{attribute 'linkalways'} 
{attribute 'no_explicit_call' := 'This FB is a CLASS and must be accessed using methods or properties'}
{attribute 'enable_dynamic_creation'}
FUNCTION_BLOCK ResetGroupCommand EXTENDS NciCommand
VAR
	_fb : CfgReconfigGroup;
	_groupId : UDINT;
	_timeout : TIME;
END_VAR

METHOD FB_init : BOOL
VAR_INPUT
	bInitRetains : BOOL; // if TRUE, the retain variables are initialized (warm start / cold start)
	bInCopyCode : BOOL;  // if TRUE, the instance afterwards gets moved into the copy code (online change)
	nci : I_Nci;
	timeout : TIME;
END_VAR
IF nci <> 0 THEN
	_groupId := nci.GroupId;
END_IF
_timeout := timeout;
END_METHOD

METHOD PROTECTED  WhileBusy
VAR_INPUT
	CommandState : I_CommandBusyState;
END_VAR
_fb(
	bExecute := TRUE,
	nGroupId := _groupId,
	tTimeOut := _timeout
);

IF _fb.bBusy THEN
	RETURN;
END_IF

IF _fb.bErr THEN
	_fb(bExecute := FALSE);
	CommandState.SetError(_fb.nErrId);
	RETURN;
END_IF

_fb(bExecute := FALSE);
CommandState.SetDone();
END_METHOD

END_FUNCTION_BLOCK

(* stored: Version 1.1.0.1, ProductVersion 3.1.4024.12
   POU ResetGroupCommand: Id {d4defed5-a731-40bc-8b88-b0e450582365}, SpecialFunc None
   Method FB_init: Id {c5637d5b-b1fe-452e-a302-54ee7e177d31}
   Method WhileBusy: Id {7806ec84-349c-4aa7-943c-7bd1a08a1af2} *)
